// TIA Portal V20 export
TYPE "LKinCtrl_typePnPLinPointParameter"
   STRUCT
      usePoint : Bool;   // Use or ignore point
      position : Array[1..6] of LReal;   // Cartesian position
      coordSystem : DInt;   // 0: WCS; 1: OCS[1]; 2: OCS[2]; 3: OCS[3]; 100: MCS
      bufferMode : DInt := 1;   // bufferMode for path motion
      transitionParameter : Array[1..5] of LReal;   // transitionParameter for path motion
      tracking : "LKinCtrl_typePnPTrackingProperties";   // Tracking properties
      directionA : DInt := 3;   // 1 - positive, 2 - negative, 3 - shortest way (Only necessary up to 4D Kinematics)
      pathDynamics : "LKinCtrl_typePathDynamics";   // Path dynamics specification
      dynamicAdaption : DInt;   // 0=no dynamic adaption, 1=dynamic adaptation with segmentation of the path, 2=dynamic adaptation without segmentation of the path
      distanceToPrevious : LReal;   // Linear distance to previous point
   END_STRUCT;
   // transitionParameter[1] := -1.0;
END_TYPE
